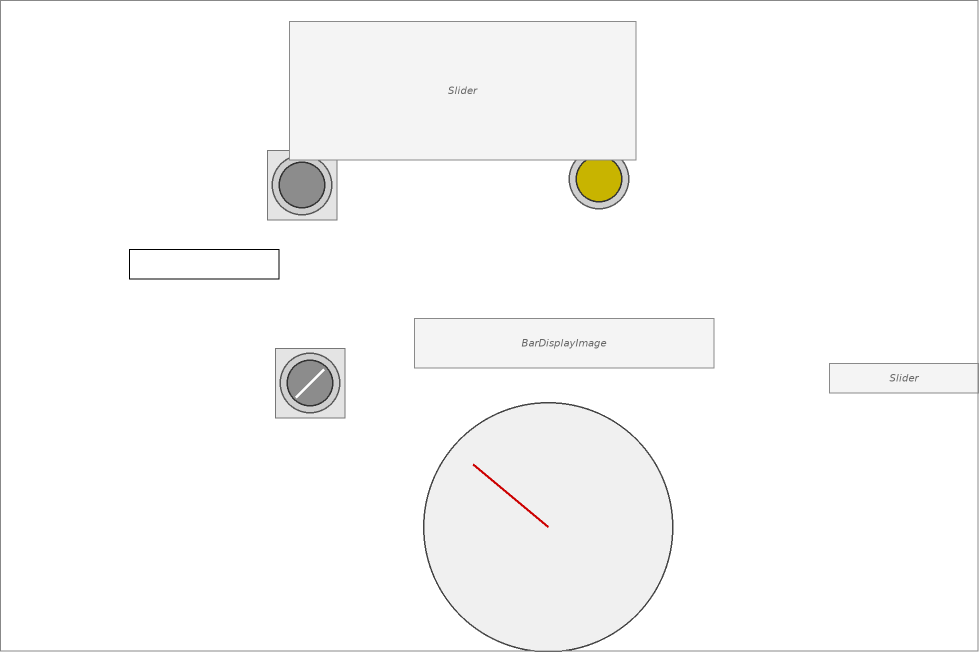
VISUALIZATION Visualization  // 979x652
    Lamp1 (564,144 70x70), variable: MAIN.bLamp, style: Lamp-Lamp1-Yellow
    PushSwitchLed (267,150 70x70), variable: MAIN.btimer_start, behaviour: TOGGLE, style: Switch-PushSwitchLed-Gray
    RotarySwitch (275,348 70x70), behaviour: TOGGLE, style: Switch-RotarySwitch-Gray
    BarDisplayImage (414,318 300x50), value: MAIN.iCounter, style: BarDisplayImage-Gray, scale format: %.1f, scale 0..100
    Meter180 (423,402 250x250), style: Meter-Meter180-Gray, scale format: %.1f, scale 0..100
    Rectangle (129,249 150x30)
    Slider (289,21 347x139), scale 0..1200
    Slider (829,363 150x30), scale 0..100
END_VISUALIZATION

(* stored: Version 1.1.0.1, ProductVersion 3.1.4024.13
   Visu Visualization: Id {2c64a80c-b703-4853-bc40-3ed8e3214e36} *)
